// TIA Portal V18 export
VAR_GLOBAL   // PLC tag table "RemoteIO_DI_2"
   "iH-shaftLoadingDetection1" AT %I2000.0 : Bool;   // H-shaft上料线体料盘检测光电1
   "iH-shaftLoadingDetection2" AT %I2000.1 : Bool;   // H-shaft上料线体料盘检测光电2
   "iH-shaftLoadingDetection3" AT %I2000.2 : Bool;   // H-shaft上料线体料盘检测光电3
   "iH-shaftLoadingDetection4" AT %I2000.3 : Bool;   // H-shaft上料线体料盘检测光电4
   "H-shaftPalletEmptyCheck1" AT %I2000.4 : Bool;   // 备用_I2000.4
   "H-shaftPalletEmptyCheck2" AT %I2000.5 : Bool;   // 备用_I2000.5
   "H-shaftPalletEmptyCheck3" AT %I2000.6 : Bool;   // 备用_I2000.6
   "iH-shaftPalletEmptyCheck4" AT %I2000.7 : Bool;   // 备用_I2000.7
   "iH-shaftTakeDetection1" AT %I2001.0 : Bool;   // H-shaft取空盘料盘检测光电1
   "iH-shaftTakeDetection2" AT %I2001.1 : Bool;   // H-shaft取空盘料盘检测光电2
   "iH-shaftTakeDetection3" AT %I2001.2 : Bool;   // H-shaft取空盘料盘检测光电3
   "iH-shaftTakeShaftDetection" AT %I2001.3 : Bool;   // H-shaft取空盘shaft空盘有无检测
   "iH-shaftTakeGateDetection" AT %I2001.4 : Bool;   // H-shaft取空盘抽屉门到位检测
   "RESERVE_I2001.5" AT %I2001.5 : Bool;   // 备用_I2001.5
   "RESERVE_I2001.6" AT %I2001.6 : Bool;   // 备用_I2001.6
   "RESERVE_I2001.7" AT %I2001.7 : Bool;   // 备用_I2001.7
   "iH-shaftLiftingPalletLocationCylinderInWP" AT %I2002.0 : Bool;   // H-shaft 顶升位托盘定位气缸工作位
   "iH-shaftLiftingPalletLocationCylinderInHP" AT %I2002.1 : Bool;   // H-shaft 顶升位托盘定位气缸原始位
   "iH-shaftLiftingLiftingCylinderInWP" AT %I2002.2 : Bool;   // H-shaft 顶升位顶升气缸工作位
   "iH-shaftLiftingLiftingCylinderInHP" AT %I2002.3 : Bool;   // H-shaft 顶升位顶升气缸原始位
   "iH-shaftLiftingPalletIn" AT %I2002.4 : Bool;   // H-shaft 顶升位托盘到位检测
   "iH-shaftLiftingPalletDischarge" AT %I2002.5 : Bool;   // H-shaft 顶升位托盘出料检测
   "iH-shaftMiddleDetection" AT %I2002.6 : Bool;   // 备用_I2002.6
   "RESERVE_I2002.7" AT %I2002.7 : Bool;   // 备用_I2002.7
   "iJ-magnetLoadingDetection1" AT %I2003.0 : Bool;   // J-magnet上料线体料盘检测光电1
   "iJ-magnetLoadingDetection2" AT %I2003.1 : Bool;   // J-magnet上料线体料盘检测光电2
   "iJ-magnetLoadingDetection3" AT %I2003.2 : Bool;   // J-magnet上料线体料盘检测光电3
   "iJ-magnetLoadingDetection4" AT %I2003.3 : Bool;   // J-magnet上料线体料盘检测光电4
   "J-mganePalletEmptyCheck1" AT %I2003.4 : Bool;   // 备用_I2003.4
   "J-mganePalletEmptyCheck2" AT %I2003.5 : Bool;   // 备用_I2003.5
   "J-mganePalletEmptyCheck3" AT %I2003.6 : Bool;   // 备用_I2003.6
   "J-mganePalletEmptyCheck4" AT %I2003.7 : Bool;   // 备用_I2003.7
   "iJ-magnetTakeDetection1" AT %I2004.0 : Bool;   // J-magnet取空盘料盘检测光电1
   "iJ-magnetTakeDetection2" AT %I2004.1 : Bool;   // J-magnet取空盘料盘检测光电2
   "iJ-magnetTakeDetection3" AT %I2004.2 : Bool;   // J-magnet取空盘料盘检测光电3
   "iJ-magnetTakeShaftDetection" AT %I2004.3 : Bool;   // J-magnet取空盘shaft空盘有无检测
   "iJ-magnetTakeGateDetection" AT %I2004.4 : Bool;   // J-magnet取空盘抽屉门到位检测
   "RESERVE_I2004.5" AT %I2004.5 : Bool;   // 备用_I2004.5
   "RESERVE_I2004.6" AT %I2004.6 : Bool;   // 备用_I2004.6
   "RESERVE_I2004.7" AT %I2004.7 : Bool;   // 备用_I2004.7
   "iJ-magnetLiftingPalletLocationCylinderInWP" AT %I2005.0 : Bool;   // J-magnet 顶升托盘定位气缸工作位
   "iJ-magnetLiftingPalletLocationCylinderInHP" AT %I2005.1 : Bool;   // J-magnet 顶升托盘定位气缸原始位
   "iJ-magnetLiftingLiftingCylinderInWP" AT %I2005.2 : Bool;   // J-magnet 顶升顶升气缸工作位
   "iJ-magnetLiftingLiftingCylinderInHP" AT %I2005.3 : Bool;   // J-magnet 顶升顶升气缸原始位
   "iJ-magnetLiftingPalletInPlaceDetection" AT %I2005.4 : Bool;   // J-magnet 顶升托盘到位检测
   "iJ-magnetLiftingPalletDischargeDetection" AT %I2005.5 : Bool;   // J-magnet 顶升托盘出料检测
   "iJ-MagnetMiddleDetection" AT %I2005.6 : Bool;   // 备用_I2005.6
   "RESERVE_I2005.7" AT %I2005.7 : Bool;   // 备用_I2005.7
   "iK-reserveLoadingDetection1" AT %I2006.0 : Bool;   // K-预留上料线体料盘检测光电1
   "iK-reserveLoadingDetection2" AT %I2006.1 : Bool;   // K-预留上料线体料盘检测光电2
   "iK-reserveLoadingDetection3" AT %I2006.2 : Bool;   // K-预留上料线体料盘检测光电3
   "iK-reserveLoadingDetection4" AT %I2006.3 : Bool;   // K-预留上料线体料盘检测光电4
   "K-reservePalletEmptyCheck1" AT %I2006.4 : Bool;   // 备用_I2006.4
   "K-reservePalletEmptyCheck2" AT %I2006.5 : Bool;   // 备用_I2006.5
   "K-reservePalletEmptyCheck3" AT %I2006.6 : Bool;   // 备用_I2006.6
   "K-reservePalletEmptyCheck4" AT %I2006.7 : Bool;   // 备用_I2006.7
   "RESERVE_I2007.0" AT %I2007.0 : Bool;
   "RESERVE_I2007.1" AT %I2007.1 : Bool;
   "RESERVE_I2007.2" AT %I2007.2 : Bool;
   "RESERVE_I2007.3" AT %I2007.3 : Bool;
   "RESERVE_I2007.4" AT %I2007.4 : Bool;
   "RESERVE_I2007.5" AT %I2007.5 : Bool;
   "RESERVE_I2007.6" AT %I2007.6 : Bool;
   "RESERVE_I2007.7" AT %I2007.7 : Bool;
   "iK-reserveTakeDetection1" AT %I2008.0 : Bool;   // K-预留取空盘料盘检测光电1
   "iK-reserveTakeDetection2" AT %I2008.1 : Bool;   // K-预留取空盘料盘检测光电2
   "iK-reserveTakeDetection3" AT %I2008.2 : Bool;   // K-预留取空盘料盘检测光电3
   "iK-reserveTakeShaftDetection" AT %I2008.3 : Bool;   // K-预留取空盘shaft空盘有无检测
   "iK-reserveTakeGateDetection" AT %I2008.4 : Bool;   // K-预留取空盘抽屉门到位检测
   "RESERVE_I2008.5" AT %I2008.5 : Bool;   // 备用_I2008.5
   "RESERVE_I2008.6" AT %I2008.6 : Bool;   // 备用_I2008.6
   "RESERVE_I2008.7" AT %I2008.7 : Bool;   // 备用_I2008.7
   "iK-reserveLifting3PalletLocationCylinderInWP" AT %I2100.0 : Bool;   // K-预留顶升位3托盘定位气缸工作位
   "iK-reserveLifting3PalletLocationCylinderInHP" AT %I2100.1 : Bool;   // K-预留顶升位3托盘定位气缸原始位
   "iK-reserveLifting3LiftingCylinderInWP" AT %I2100.2 : Bool;   // K-预留顶升位3顶升气缸工作位
   "iK-reserveLifting3LiftingCylinderInHP" AT %I2100.3 : Bool;   // K-预留顶升位3顶升气缸原始位
   "iK-reserveLifting3PalletInPlaceDetection" AT %I2100.4 : Bool;   // K-预留顶升位3托盘到位检测
   "iK-reserveLifting3PalletDischargeDetection" AT %I2100.5 : Bool;   // K-预留顶升位3托盘出料检测
   "iK-reserveMiddleDetection" AT %I2100.6 : Bool;   // 备用_I2100.6
   "RESERVE_I2100.7" AT %I2100.7 : Bool;   // 备用_I2100.7
   "RESERVE_I2101.0" AT %I2101.0 : Bool;
   "RESERVE_I2101.1" AT %I2101.1 : Bool;
   "RESERVE_I2101.2" AT %I2101.2 : Bool;
   "RESERVE_I2101.3" AT %I2101.3 : Bool;
   "RESERVE_I2101.4" AT %I2101.4 : Bool;
   "RESERVE_I2101.5" AT %I2101.5 : Bool;
   "RESERVE_I2101.6" AT %I2101.6 : Bool;
   "RESERVE_I2101.7" AT %I2101.7 : Bool;
   "iL-UnloadingDetection1" AT %I2102.0 : Bool;   // L-下料线体料盘检测光电1
   "iL-UnloadingDetection2" AT %I2102.1 : Bool;   // L-下料线体料盘检测光电2
   "iL-UnloadingDetection3" AT %I2102.2 : Bool;   // L-下料线体料盘检测光电3
   "L-UnloadinPalletEmptyCheck1" AT %I2102.3 : Bool;   // 备用_I2102.3
   "L-UnloadinPalletEmptyCheck2" AT %I2102.4 : Bool;   // 备用_I2102.4
   "L-UnloadinPalletEmptyCheck3" AT %I2102.5 : Bool;   // 备用_I2102.5
   "L-UnloadinTakeGateDetection" AT %I2102.6 : Bool;   // 备用_I2102.6
   "RESERVE_I2102.7" AT %I2102.7 : Bool;   // 备用_I2102.7
   "RESERVE_I2103.0" AT %I2103.0 : Bool;
   "RESERVE_I2103.1" AT %I2103.1 : Bool;
   "RESERVE_I2103.2" AT %I2103.2 : Bool;
   "RESERVE_I2103.3" AT %I2103.3 : Bool;
   "RESERVE_I2103.4" AT %I2103.4 : Bool;
   "RESERVE_I2103.5" AT %I2103.5 : Bool;
   "RESERVE_I2103.6" AT %I2103.6 : Bool;
   "RESERVE_I2103.7" AT %I2103.7 : Bool;
   "iL-UnloadingTransPalletLocationCylinderInWP" AT %I2104.0 : Bool;   // L-下料线体移栽托盘定位气缸工作位
   "iL-UnloadingTransPalletLocationCylinderInHP" AT %I2104.1 : Bool;   // L-下料线体移栽托盘定位气缸原始位
   "iL-UnloadingTransCylinderInWP" AT %I2104.2 : Bool;   // L-下料线体移栽气缸工作位
   "iL-UnloadingTransCylinderInHP" AT %I2104.3 : Bool;   // L-下料线体移栽气缸原始位
   "iL-UnloadingTransplantingPalletInPlaceDetection" AT %I2104.4 : Bool;   // L-下料线体移栽托盘到位检测
   "iL-UnloadingPalletDischargeDetection" AT %I2104.5 : Bool;   // L-下料线体托盘出料检测
   "RESERVE_I2104.6" AT %I2104.6 : Bool;   // 备用_I2104.6
   "RESERVE_I2104.7" AT %I2104.7 : Bool;   // 备用_I2104.7
END_VAR
